(* CoDeSys 2.3 export: GVL_SUBSCRIPTION.EXP *)

(* Global variable list: AdsClientTests/GVL_Subscription *)
VAR_GLOBAL
	NumericValue_10ms		 : INT;
	NumericValue_100ms 		: INT;
	NumericValue_1000ms 	: INT;
	Numericvalue_Constant	: INT := 12245;
END_VAR
